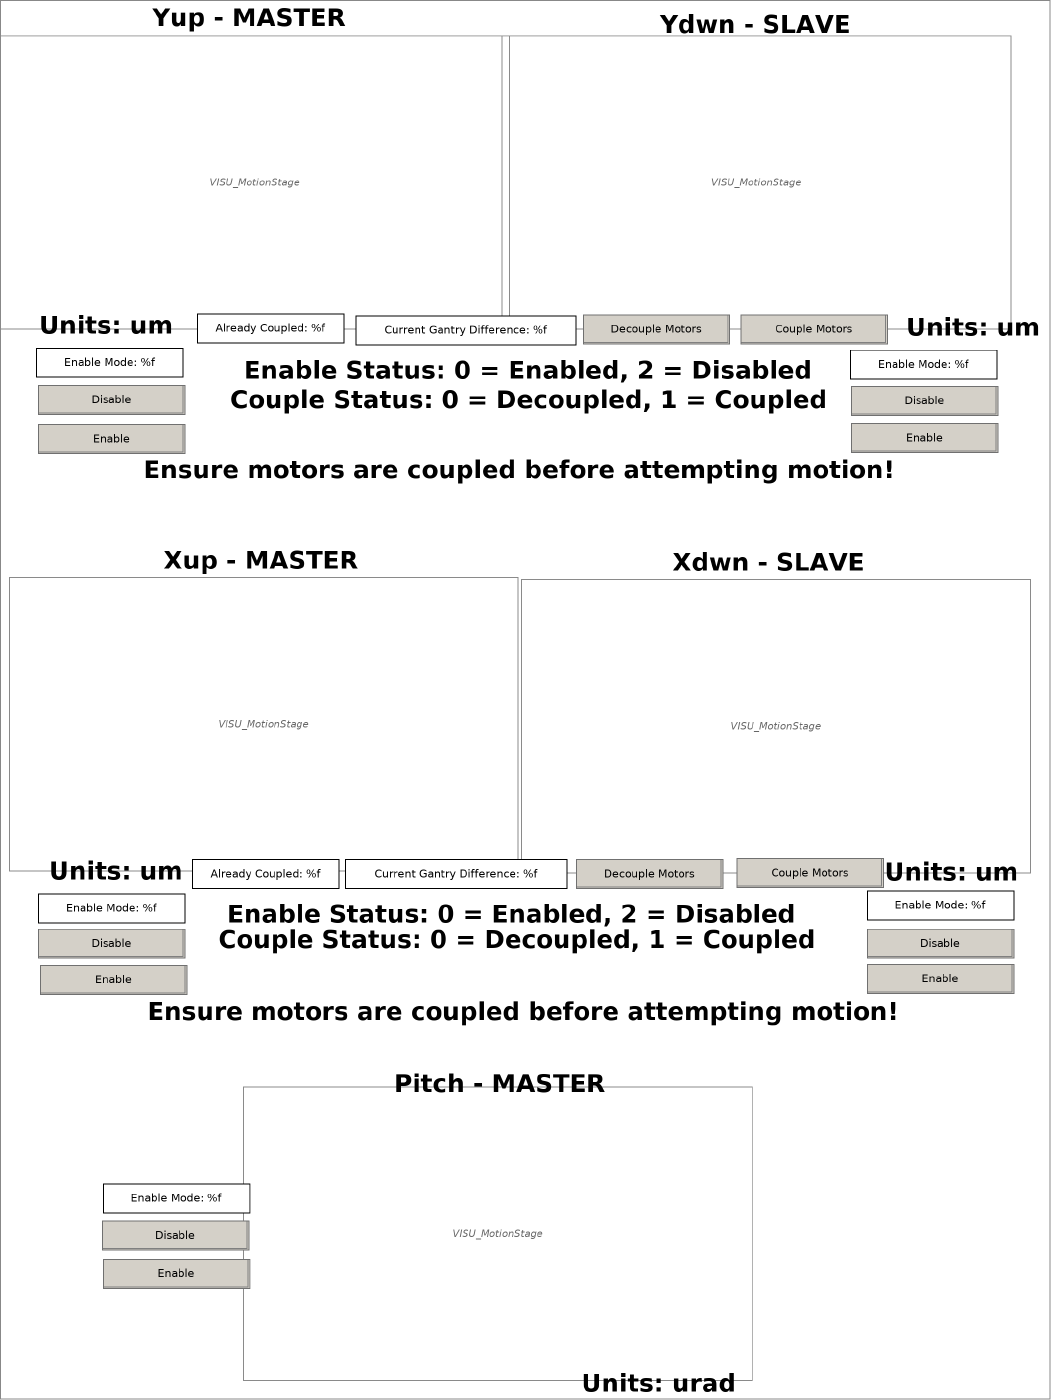
VISUALIZATION Visualization  // 1073x1429
    Label (14,2 481x31), "Yup - MASTER"
    Frame (0,36 520x300)
        shows VISU_MotionStage(VisuMotionStage := MAIN.M1, Extras := MAIN.M1_Extras)
    Frame (512,36 520x300)
        shows VISU_MotionStage(VisuMotionStage := MAIN.M2, Extras := MAIN.M2_Extras)
    Label (531,9 481x31), "Ydwn - SLAVE"
    Rectangle (201,320 150x30), "Already Coupled: %f", tooltip "Couple Status: TRUE if coupled", text variable: MAIN.bGantryAlreadyCoupledY
    Rectangle (363,322 225x30), "Current Gantry Difference: %f", tooltip "Current Gantry Difference in um", text variable: MAIN.fCurrGantryY_um
    Button (756,321 150x30), "Couple Motors", tooltip "Press To Couple Motors", text variable: MAIN.bExecuteCoupleY
        OnMouseDown: execute { MAIN.bExecuteCoupleY := TRUE; }
    Frame (9,589 520x300)
        shows VISU_MotionStage(VisuMotionStage := MAIN.M3, Extras := MAIN.M3_Extras)
    Label (26,556 481x31), "Xup - MASTER"
    Frame (532,591 520x300)
        shows VISU_MotionStage(VisuMotionStage := MAIN.M4, Extras := MAIN.M4_Extras)
    Label (544,558 481x31), "Xdwn - SLAVE"
    Rectangle (196,877 150x30), "Already Coupled: %f", tooltip "Couple Status: TRUE if coupled", text variable: MAIN.bGantryAlreadyCoupledX
    Rectangle (352,877 227x30), "Current Gantry Difference: %f", tooltip "Current Gantry Difference in um", text variable: MAIN.fCurrGantryX_um
    Frame (248,1109 520x300)
        shows VISU_MotionStage(VisuMotionStage := MAIN.M5, Extras := MAIN.M5_Extras)
    Label (270,1090 481x31), "Pitch - MASTER"
    Label (31,316 155x31), "Units: um"
    Label (916,318 155x31), "Units: um"
    Label (41,873 155x31), "Units: um"
    Label (894,874 155x31), "Units: um"
    Label (595,1396 155x31), "Units: urad"
    Rectangle (37,355 150x30), "Enable Mode: %f", tooltip "Write 0 to Enable, 2 to Disable", text variable: MAIN.M1.nEnableMode
    Rectangle (868,357 150x30), "Enable Mode: %f", tooltip "Write 0 to Enable, 2 to Disable", text variable: MAIN.M2.nEnableMode
    Button (595,321 150x30), "Decouple Motors", tooltip "Press To Decouple Motors for independent control"
        OnMouseDown: execute { MAIN.bExecuteDecoupleY := TRUE; }
    Button (39,393 150x30), "Disable"
        OnMouseDown: execute { MAIN.M1.nEnableMode := 2; }
    Button (39,433 150x30), "Enable", colour toggle: MAIN.bExecuteDecoupleY
        OnMouseDown: execute { MAIN.M1.nEnableMode := 0; }
    Button (869,394 150x30), "Disable"
        OnMouseDown: execute { MAIN.M2.nEnableMode := 2; }
    Button (869,432 150x30), "Enable", colour toggle: MAIN.bExecuteDecoupleY
        OnMouseDown: execute { MAIN.M2.nEnableMode := 0; }
    Button (588,877 150x30), "Decouple Motors", tooltip "Press To Decouple Motors for independent control"
        OnMouseDown: execute { MAIN.bExecuteDecoupleX := TRUE; }
    Button (752,876 150x30), "Couple Motors", tooltip "Press To Couple Motors", text variable: MAIN.bExecuteCoupleY
        OnMouseDown: execute { MAIN.bExecuteCoupleX := TRUE; }
    Rectangle (39,912 150x30), "Enable Mode: %f", tooltip "Write 0 to Enable, 2 to Disable", text variable: MAIN.M3.nEnableMode
    Button (39,948 150x30), "Disable"
        OnMouseDown: execute { MAIN.M3.nEnableMode := 2; }
    Button (41,985 150x30), "Enable", colour toggle: MAIN.bExecuteDecoupleY
        OnMouseDown: execute { MAIN.M3.nEnableMode := 0; }
    Rectangle (885,909 150x30), "Enable Mode: %f", tooltip "Write 0 to Enable, 2 to Disable", text variable: MAIN.M4.nEnableMode
    Button (885,948 150x30), "Disable"
        OnMouseDown: execute { MAIN.M4.nEnableMode := 2; }
    Button (885,984 150x30), "Enable", colour toggle: MAIN.bExecuteDecoupleY
        OnMouseDown: execute { MAIN.M4.nEnableMode := 0; }
    Rectangle (105,1208 150x30), "Enable Mode: %f", tooltip "Write 0 to Enable, 2 to Disable", text variable: MAIN.M5.nEnableMode
    Button (104,1246 150x30), "Disable"
        OnMouseDown: execute { MAIN.M5.nEnableMode := 2; }
    Button (105,1285 150x30), "Enable", colour toggle: MAIN.bExecuteDecoupleY
        OnMouseDown: execute { MAIN.M5.nEnableMode := 0; }
    Label (255,362 568x31), "Enable Status: 0 = Enabled, 2 = Disabled"
    Label (247,392 586x31), "Couple Status: 0 = Decoupled, 1 = Coupled"
    Label (238,917 568x31), "Enable Status: 0 = Enabled, 2 = Disabled"
    Label (235,943 586x31), "Couple Status: 0 = Decoupled, 1 = Coupled"
    Label (150,464 760x30), "Ensure motors are coupled before attempting motion!"
    Label (154,1017 760x30), "Ensure motors are coupled before attempting motion!"
END_VISUALIZATION

(* stored: Version 1.1.0.1, ProductVersion 3.1.4022.18
   Visu Visualization: Id {af2f16f4-e7e7-4019-a84a-cc323e4115d2} *)
